FUNCTION_BLOCK FB_ReadTextList
VAR_INPUT
	iTargetfilestring:STRING(255):= 'C:\PLC\Messages\FileName.XML'; // 'C:\PLC\Messages\Mc_Alarms.XML'
	iStart: BOOL;
	iReset: BOOL;


END_VAR
VAR_OUTPUT
	theemessage:string(255);
	outindex:INT;
	

END_VAR

VAR_OUTPUT
fHandle:UINT;
END_VAR


VAR
	
	openfileee: FB_FileOpen;
	openfileee2: FB_FileOpen;
	openTheFile: BOOL;
	gettaTheFile: FB_FileGets;
	gettaTheFile2: FB_FileGets;
	readatheFile: BOOL;
	textListNameLocation: INT;
	findText: FB_FindTextIndexNum;
	findLangText: FB_FindTextLangText;
	examplestring: STRING(255);
	tResetFunc: BOOL;
	fileNumber: UINT;
	fileisEOF: BOOL;
	closeatheFile: FB_FileClose;
	IsCorrectLineForText: INT;
	isCorrectLine: BOOL;
END_VAR
//theme:8b5rIFci5vs
VAR // added by the converter: edge detectors and wires of the graphical bodies
    _rt1, _rt2, _rt3, _rt4, _rt5, _rt6, _rt7, _rt8 : R_TRIG;
    _w1, _w2, _w3, _w4, _w5 : BOOL;
END_VAR

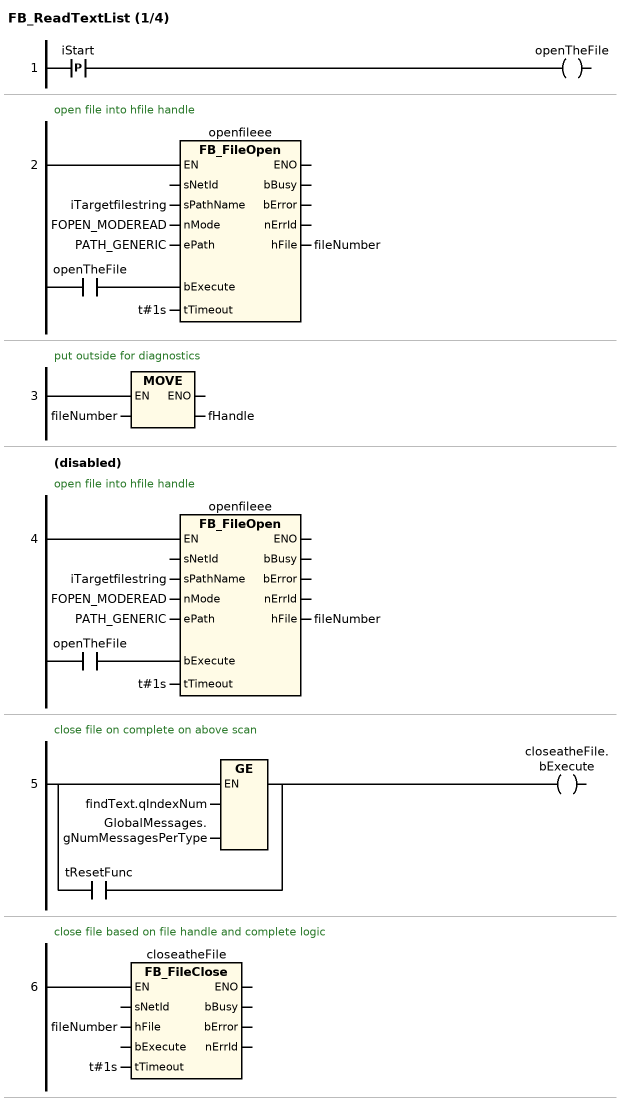
// NETWORK 1
_rt1(CLK := iStart);
openTheFile := _rt1.Q;

// NETWORK 2
// open file into hfile handle
openfileee(
    sPathName := iTargetfilestring,
    nMode := FOPEN_MODEREAD,
    ePath := PATH_GENERIC,
    bExecute := openTheFile,
    tTimeout := t#1s,
    hFile => fileNumber); // FB_FileOpen

// NETWORK 3
// put outside for diagnostics
fHandle := fileNumber;

// NETWORK 4 (disabled)
// open file into hfile handle
// openfileee(
//     sPathName := iTargetfilestring,
//     nMode := FOPEN_MODEREAD,
//     ePath := PATH_GENERIC,
//     bExecute := openTheFile,
//     tTimeout := t#1s,
//     hFile => fileNumber); // FB_FileOpen

// NETWORK 5
// close file on complete on above scan
_w1 := tResetFunc;
IF NOT _w1 THEN
    _w1 := findText.qIndexNum >= GlobalMessages.gNumMessagesPerType;
END_IF
closeatheFile.bExecute := _w1;

// NETWORK 6
// close file based on file handle and complete logic
closeatheFile(hFile := fileNumber, tTimeout := t#1s); // FB_FileClose

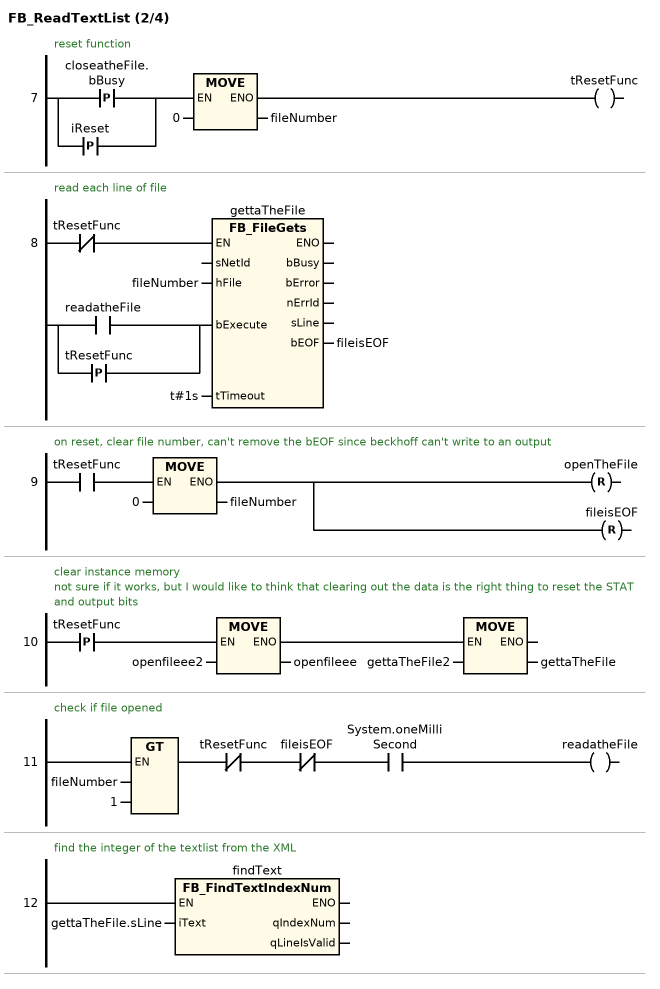
// NETWORK 7
// reset function
_rt2(CLK := closeatheFile.bBusy);
_rt3(CLK := iReset);
_w2 := _rt2.Q OR _rt3.Q;
IF _w2 THEN fileNumber := 0; END_IF
tResetFunc := _w2;

// NETWORK 8
// read each line of file
_rt4(CLK := tResetFunc);
IF NOT tResetFunc THEN
    gettaTheFile(hFile := fileNumber, bExecute := readatheFile OR _rt4.Q, tTimeout := t#1s, bEOF => fileisEOF); // FB_FileGets
END_IF

// NETWORK 9
// on reset, clear file number, can't remove the bEOF since beckhoff can't write to an output
_w3 := tResetFunc;
IF _w3 THEN fileNumber := 0; END_IF
openTheFile R= _w3;
fileisEOF R= _w3;

// NETWORK 10
// clear instance memory
// not sure if it works, but I would like to think that clearing out the data is the right thing to reset the STAT and output bits
_rt5(CLK := tResetFunc);
_w4 := _rt5.Q;
IF _w4 THEN openfileee := openfileee2; END_IF
IF _w4 THEN gettaTheFile := gettaTheFile2; END_IF

// NETWORK 11
// check if file opened
readatheFile := fileNumber > 1 AND NOT tResetFunc AND NOT fileisEOF AND System.oneMilliSecond;

// NETWORK 12
// find the integer of the textlist from the XML
findText(iText := gettaTheFile.sLine); // FB_FindTextIndexNum

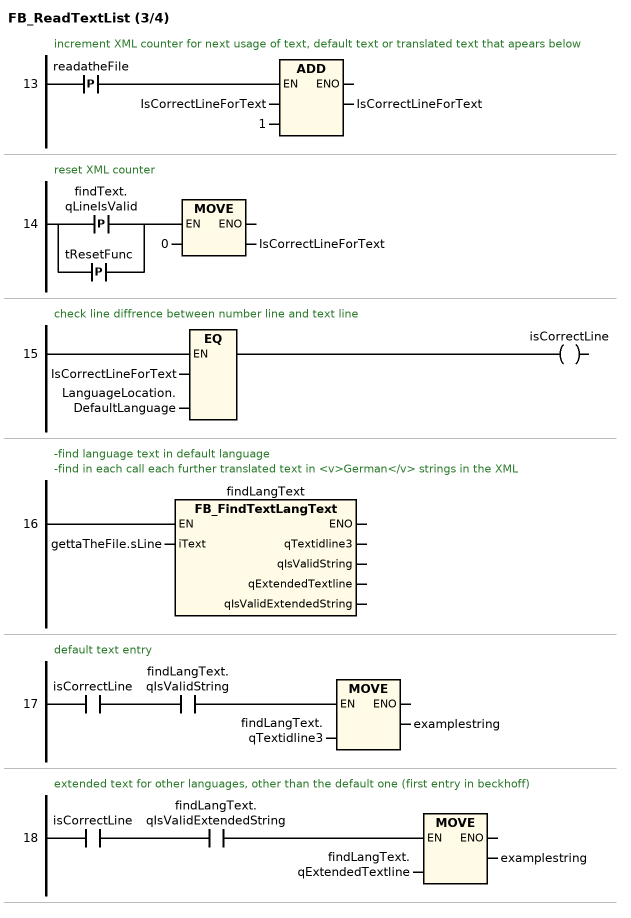
// NETWORK 13
// increment XML counter for next usage of text, default text or translated text that apears below
_rt6(CLK := readatheFile);
IF _rt6.Q THEN IsCorrectLineForText := IsCorrectLineForText + 1; END_IF

// NETWORK 14
// reset XML counter
_rt7(CLK := findText.qLineIsValid);
_rt8(CLK := tResetFunc);
IF _rt7.Q OR _rt8.Q THEN IsCorrectLineForText := 0; END_IF

// NETWORK 15
// check line diffrence between number line and text line
isCorrectLine := IsCorrectLineForText = LanguageLocation.DefaultLanguage;

// NETWORK 16
// -find language text in default language
// -find in each call each further translated text in <v>German</v> strings in the XML
findLangText(iText := gettaTheFile.sLine); // FB_FindTextLangText

// NETWORK 17
// default text entry
IF isCorrectLine AND findLangText.qIsValidString THEN examplestring := findLangText.qTextidline3; END_IF

// NETWORK 18
// extended text for other languages, other than the default one (first entry in beckhoff)
IF isCorrectLine AND findLangText.qIsValidExtendedString THEN
    examplestring := findLangText.qExtendedTextline;
END_IF

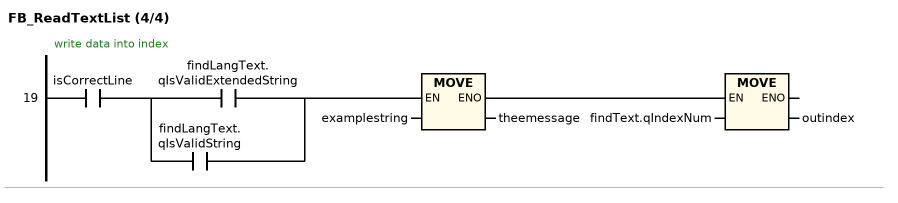
// NETWORK 19
// write data into index
_w5 := isCorrectLine AND (findLangText.qIsValidExtendedString OR findLangText.qIsValidString);
IF _w5 THEN theemessage := examplestring; END_IF
IF _w5 THEN outindex := findText.qIndexNum; END_IF

END_FUNCTION_BLOCK

(* stored: Version 1.1.0.1, ProductVersion 3.1.4024.12
   POU FB_ReadTextList: Id {65e74b11-869a-49fe-b59c-ddf45ba61820}, SpecialFunc None *)
